SYSTEM Test_RMTDev (* System Configuration *)
  (* Standard: 61499-1 *)
  (* Version 0.3, 2003-12-05, JHC, Rockwell Automation, Renamed from NEWSYSTEM. *)
  (* Version 0.2, 2002-11-05, JHC, Rockwell Automation, Fixed missing (empty) FBD in Application. *)
  (* Version 0.1, 2002-01-17, JHC, Rockwell Automation, Minor cleanup *)
  (* Version 0.0, 2000-05-27, JHC, Rockwell Automation *)
  APPLICATION APP1
  END_APPLICATION
  DEVICE DEV1 : FRAME_DEVICE
    RESOURCE RES1 : PANEL_RESOURCE
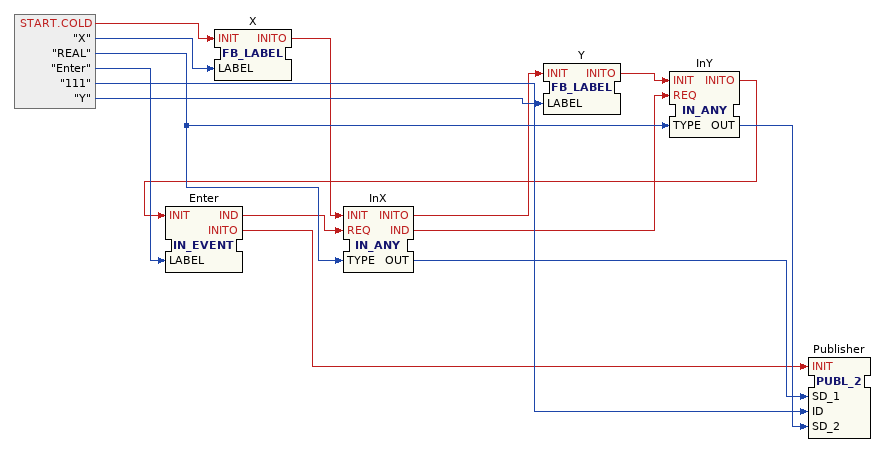
      FBS
        X : FB_LABEL;
        InX : IN_ANY;
        Enter : IN_EVENT;
        Publisher : PUBL_2;
        Y : FB_LABEL;
        InY : IN_ANY;
      END_FBS
      EVENT_CONNECTIONS
        START.COLD TO X.INIT;
        X.INITO TO InX.INIT;
        InX.INITO TO Y.INIT;
        Y.INITO TO InY.INIT;
        InY.INITO TO Enter.INIT;
        Enter.IND TO InX.REQ;
        InX.IND TO InY.REQ;
        Enter.INITO TO Publisher.INIT;
      END_CONNECTIONS
      DATA_CONNECTIONS
        "X" TO X.LABEL;
        "REAL" TO InX.TYPE;
        "Enter" TO Enter.LABEL;
        InX.OUT TO Publisher.SD_1;
        "111" TO Publisher.ID;
        "Y" TO Y.LABEL;
        "REAL" TO InY.TYPE;
        InY.OUT TO Publisher.SD_2;
      END_CONNECTIONS
    END_RESOURCE
  END_DEVICE
  DEVICE Ausgabe : RMT_DEV
    RESOURCE FOO : PANEL_RESOURCE
    END_RESOURCE
  END_DEVICE
  DATA_CONNECTIONS (* parameter values *)
    [0,0,150,250] TO DEV1.BOUNDS;
    [0,1] TO DEV1.GRID;
  END_CONNECTIONS
END_SYSTEM
